// TIA Portal V16 export
ORGANIZATION_BLOCK "Main"   // OB1, LAD, ProgramCycle
{ S7_Optimized_Access := 'TRUE' }
// stored: AutoNumber false
   VAR_INPUT
      Initial_Call : Bool;
      Remanence : Bool;
   END_VAR
BEGIN

REGION Network 1: Conveyor control - cyclic LAD call
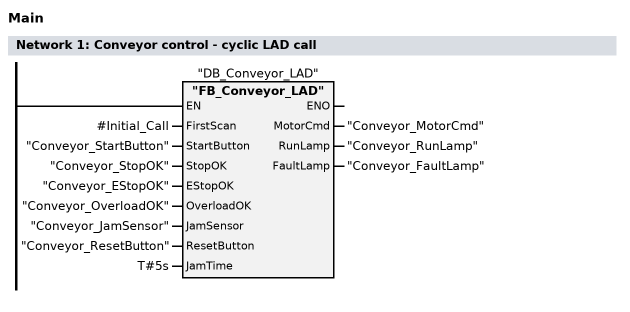
   RUNG wire#powerrail
      "DB_Conveyor_LAD"(FirstScan := #Initial_Call, StartButton := "Conveyor_StartButton", StopOK := "Conveyor_StopOK", EStopOK := "Conveyor_EStopOK", OverloadOK := "Conveyor_OverloadOK", JamSensor := "Conveyor_JamSensor", ResetButton := "Conveyor_ResetButton", JamTime := T#5s, MotorCmd => "Conveyor_MotorCmd", RunLamp => "Conveyor_RunLamp", FaultLamp => "Conveyor_FaultLamp")
   END_RUNG
   // the same network as SCL:
   "DB_Conveyor_LAD"(FirstScan := #Initial_Call,   // "FB_Conveyor_LAD"
                     StartButton := "Conveyor_StartButton",
                     StopOK := "Conveyor_StopOK",
                     EStopOK := "Conveyor_EStopOK",
                     OverloadOK := "Conveyor_OverloadOK",
                     JamSensor := "Conveyor_JamSensor",
                     ResetButton := "Conveyor_ResetButton",
                     JamTime := T#5s,
                     MotorCmd => "Conveyor_MotorCmd",
                     RunLamp => "Conveyor_RunLamp",
                     FaultLamp => "Conveyor_FaultLamp");
END_REGION
END_ORGANIZATION_BLOCK
